// TwinCAT 3 PLC project drivePLC
// ProgramVersion: 3.1.4022.4
// libraries:
//   Tc2_MC2, * (Beckhoff Automation GmbH)
//   Tc2_NC, * (Beckhoff Automation GmbH)
//   Tc2_Standard, * (Beckhoff Automation GmbH)
//   Tc2_System, * (Beckhoff Automation GmbH)
//   Tc3_MC2_AdvancedHoming, * (Beckhoff Automation GmbH)
//   Tc3_Module, * (Beckhoff Automation GmbH)
//   VisuDialogs, * (System)
// project tree:
//   DUTs/ eLimitCoupling.TcDUT (not stored), eMcCommand.TcDUT (not stored), eRWParameter.TcDUT (not stored), ST_AxisControl.TcDUT, ST_MasterAxis.TcDUT (not stored), ST_MasterCoupling.TcDUT (not stored), ST_SimulateStage.TcDUT (not stored)
//   / GlobalTextList.TcGTLO, PlcTask.TcTTO, Visualization Manager.TcVMO (not stored)
//   GVLs/ GVL.TcGVL, Limits.TcGVL
//   POUs/ FB_AxisDrive.TcPOU, MAIN.TcPOU
//   VISUs/ Main.TcVIS
//   VISUs/Panels/ ButtonStates.TcTLO (not stored), CommandList.TcTLO (not stored), ImagePool.TcIPO (not stored), IO.TcVIS (not stored), SlitSet.TcVIS (not stored), Visualization.TcVIS
//   VISUs/Panels/Command VISUs/ AxisSimulation.TcVIS (not stored), Gearing.TcVIS (not stored), Homing.TcVIS (not stored), Parameters.TcVIS (not stored)
// real-time tasks:
//   TASK PlcTask: cycle T#10ms, priority 20, ADS port 350
// motion (NC):
//   TASK NC-Task 1 SAF: cycle T#2ms, priority 4, ADS port 501
//   TASK NC-Task 1 SVB: cycle T#10ms, priority 8, ADS port 511
//   AXIS North Blade (id 1)
//     Dynamic: AccelerationMaximum=5000, DecelerationMaximum=5000, Acceleration=10.7143, Deceleration=10.7143, Jerk=45.9184
//     Velo: RefSearch=1, RefSync=1, SlowManual=1, FastManual=3, Maximum=5
//     OtherSettings: AllowMotionCmdToSlave=true, DataPersistence=true, PulseDistancePos=0.1, PulseDistanceNeg=0.1
//     encoder EncType=19
//       EncPara: ScaleFactorNumerator=1, ScaleFactorDenominator=1048576, MaxCount=#xffffffff, ReferenceSystem=4
//         SoftEndMinControl: Range=-5
//         SoftEndMaxControl: Range=45
//         Inc: RefSearchInverse=true, RefSyncInverse=false, RefSoftSyncMask=#x0000ffff
//     drive DrvType=24
//       DrvPara: Inverse=true
//         Analog: VeloReferenz=5, ScaleFactorActTorque=0.1
//         TimeComp: TaskDelayCycles=1
//     controller CtrType=1
//       CtrPara: PriorControlFactor=1
//         PosDiffControl: Range=1
//         Observer: BandWidth=20
//   AXIS South Blade (id 2)
//     Dynamic: AccelerationMaximum=1500, DecelerationMaximum=1500, Acceleration=150, Deceleration=150, Jerk=225
//     Velo: RefSearch=1, RefSync=1, SlowManual=1, FastManual=3, Maximum=5
//     OtherSettings: AllowMotionCmdToSlave=true, DataPersistence=true, PulseDistancePos=0.1, PulseDistanceNeg=0.1
//     encoder EncType=19
//       EncPara: ScaleFactorNumerator=1, ScaleFactorDenominator=1048576, MaxCount=#xffffffff, ReferenceSystem=4
//         SoftEndMinControl: Range=-45
//         SoftEndMaxControl: Range=5
//         Inc: RefSoftSyncMask=#x0000ffff
//     drive DrvType=24
//       DrvPara: Inverse=true
//         Analog: VeloReferenz=5, ScaleFactorActTorque=0.1
//         TimeComp: TaskDelayCycles=1
//     controller CtrType=1
//       CtrPara: PriorControlFactor=1
//         PosDiffControl: Range=1
//         Observer: BandWidth=20
//   AXIS East Blade (id 3)
//     Dynamic: AccelerationMaximum=1500, DecelerationMaximum=1500, Acceleration=150, Deceleration=150, Jerk=225
//     Velo: RefSearch=1, RefSync=1, SlowManual=1, FastManual=3, Maximum=5
//     OtherSettings: AllowMotionCmdToSlave=true, DataPersistence=true, PulseDistancePos=0.1, PulseDistanceNeg=0.1
//     encoder EncType=19
//       EncPara: ScaleFactorNumerator=1, ScaleFactorDenominator=1048576, Inverse=true, MaxCount=#xffffffff, ReferenceSystem=4
//         SoftEndMinControl: Range=-5
//         SoftEndMaxControl: Range=45
//         Inc: RefSoftSyncMask=#x0000ffff
//     drive DrvType=24
//       Analog: VeloReferenz=5, ScaleFactorActTorque=0.1
//       TimeComp: TaskDelayCycles=1
//     controller CtrType=1
//       CtrPara: PriorControlFactor=1
//         PosDiffControl: Range=1
//         Observer: BandWidth=20
//   AXIS West Blade (id 4)
//     Dynamic: AccelerationMaximum=1500, DecelerationMaximum=1500, Acceleration=150, Deceleration=150, Jerk=225
//     Velo: RefSearch=1, RefSync=1, SlowManual=1, FastManual=3, Maximum=5
//     OtherSettings: AllowMotionCmdToSlave=true, DataPersistence=true, PulseDistancePos=0.1, PulseDistanceNeg=0.1
//     encoder EncType=19
//       EncPara: ScaleFactorNumerator=1, ScaleFactorDenominator=1048576, Inverse=true, MaxCount=#xffffffff, ReferenceSystem=4
//         SoftEndMinControl: Range=5
//         SoftEndMaxControl: Range=-45
//         Inc: RefSoftSyncMask=#x0000ffff
//     drive DrvType=24
//       Analog: VeloReferenz=5, ScaleFactorActTorque=0.1
//       TimeComp: TaskDelayCycles=1
//     controller CtrType=1
//       CtrPara: PriorControlFactor=1
//         Observer: BandWidth=20
//   AXIS VG (id 5)
//     Dynamic: AccelerationMaximum=200, DecelerationMaximum=200, Acceleration=150, Deceleration=150, Jerk=225
//     Velo: RefSearch=1, RefSync=1, SlowManual=1, FastManual=3, Maximum=3
//     OtherSettings: AllowMotionCmdToSlave=true, PulseDistancePos=0.1, PulseDistanceNeg=0.1
//     encoder EncType=1
//     drive DrvType=5
//       Analog: ScaleFactorActTorque=0.1
//       TimeComp: TaskDelayCycles=1
//     controller CtrType=1
//       CtrPara: PriorControlFactor=1
//         Observer: BandWidth=20
//   AXIS VC (id 6)
//     Dynamic: AccelerationMaximum=200, DecelerationMaximum=200, Acceleration=150, Deceleration=150, Jerk=225
//     Velo: RefSearch=1, RefSync=1, SlowManual=1, FastManual=3, Maximum=3
//     OtherSettings: AllowMotionCmdToSlave=true, PulseDistancePos=0.1, PulseDistanceNeg=0.1
//     encoder EncType=1
//     drive DrvType=5
//       Analog: ScaleFactorActTorque=0.1
//       TimeComp: TaskDelayCycles=1
//     controller CtrType=1
//       CtrPara: PriorControlFactor=1
//         Observer: BandWidth=20
//   AXIS HG (id 7)
//     Dynamic: AccelerationMaximum=200, DecelerationMaximum=200, Acceleration=150, Deceleration=150, Jerk=225
//     Velo: RefSearch=1, RefSync=1, SlowManual=1, FastManual=3, Maximum=3
//     OtherSettings: AllowMotionCmdToSlave=true, PulseDistancePos=0.1, PulseDistanceNeg=0.1
//     encoder EncType=1
//     drive DrvType=5
//       Analog: ScaleFactorActTorque=0.1
//       TimeComp: TaskDelayCycles=1
//     controller CtrType=1
//       CtrPara: PriorControlFactor=1
//         Observer: BandWidth=20
//   AXIS HC (id 8)
//     Dynamic: AccelerationMaximum=200, DecelerationMaximum=200, Acceleration=150, Deceleration=150, Jerk=225
//     Velo: RefSearch=1, RefSync=1, SlowManual=1, FastManual=3, Maximum=3
//     OtherSettings: AllowMotionCmdToSlave=true, PulseDistancePos=0.1, PulseDistanceNeg=0.1
//     encoder EncType=1
//     drive DrvType=5
//       Analog: ScaleFactorActTorque=0.1
//       TimeComp: TaskDelayCycles=1
//     controller CtrType=1
//       CtrPara: PriorControlFactor=1
//         Observer: BandWidth=20
// I/O:
//   DEVICE Device 1 (EtherCAT), AmsNetId 5.60.136.192.2.1
//     Term 1 (EK1200) [EK1200-5000 EtherCAT Power supply (2A E-Bus)]
//       Limits Output (EL2008) [EL2008 8Ch. Dig. Output 24V, 0.5A]
//       Limits Input (EL1008) [EL1008 8Ch. Dig. Input 24V, 3ms]
//       FB01 NORTH (EL7201) [EL7201 1Ch. MDP742 Servo motor output stage (50V, 4A)]
//       FB02 SOUTH (EL7201) [EL7201 1Ch. MDP742 Servo motor output stage (50V, 4A)]
//       FB03 EAST (EL7201) [EL7201 1Ch. MDP742 Servo motor output stage (50V, 4A)]
//       FB04 WEST (EL7201) [EL7201 1Ch. MDP742 Servo motor output stage (50V, 4A)]
//       DR01 NORTH (EL7047) [EL7047 1Ch. Stepper motor output stage (50V, 5A)]
//       DR02  SOUTH (EL7047) [EL7047 1Ch. Stepper motor output stage (50V, 5A)]
//       DR03 EAST (EL7047) [EL7047 1Ch. Stepper motor output stage (50V, 5A)]
//       DR04 WEST (EL7047) [EL7047 1Ch. Stepper motor output stage (50V, 5A)]
//       Term 21 (EL9011) [EL9011 End Terminal]
//   DEVICE Device 4 (COM Port)
// variable links:
//   NC-Task 1 SAF/Axes/East Blade <-> Device 1 (EtherCAT)/Term 1 (EK1200)/DR03 EAST (EL7047)
//     Drive/Inputs/In/nState1 @bit 3 <-> STM Status/Status/Error
//     Drive/Inputs/In/nState1 @bit 7 <-> STM Status/Status/Motor stall
//     Drive/Inputs/In/nState1 @bit 5 <-> STM Status/Status/Moving negative
//     Drive/Inputs/In/nState1 @bit 4 <-> STM Status/Status/Moving positive
//     Drive/Inputs/In/nState1 @bit 1 <-> STM Status/Status/Ready
//     Drive/Inputs/In/nState1 <-> STM Status/Status/Ready to enable
//     Drive/Inputs/In/nState1 @bit 6 <-> STM Status/Status/Torque reduced
//     Drive/Inputs/In/nState1 @bit 2 <-> STM Status/Status/Warning
//     Drive/Inputs/In/nState2 @bit 3 <-> STM Status/Status/Digital input 1
//     Drive/Inputs/In/nState2 @bit 4 <-> STM Status/Status/Digital input 2
//     Drive/Inputs/In/nState2 @bit 5 <-> STM Status/Status/Sync error
//     Drive/Inputs/In/nState2 @bit 7 <-> STM Status/Status/TxPDO Toggle
//     Drive/Inputs/In/nState4 @bit 1 <-> WcState/InputToggle
//     Drive/Inputs/In/nState4 <-> WcState/WcState
//     Drive/Outputs/Out/nCtrl1 <-> STM Control/Control/Enable
//     Drive/Outputs/Out/nCtrl1 @bit 2 <-> STM Control/Control/Reduce torque
//     Drive/Outputs/Out/nCtrl1 @bit 1 <-> STM Control/Control/Reset
//     Drive/Outputs/Out/nCtrl2 @bit 3 <-> STM Control/Control/Digital output 1
//     Drive/Outputs/Out/nDataOut2[0] <-> STM Velocity/Velocity
//   NC-Task 1 SAF/Axes/East Blade <-> Device 1 (EtherCAT)/Term 1 (EK1200)/FB03 EAST (EL7201)
//     East Bladenc/Inputs/In/nDataIn1 <-> FB Position/Position
//     East Bladenc/Inputs/In/nDcInputTime <-> InfoData/DcInputShift
//     East Bladenc/Inputs/In/nState4 @bit 1 <-> WcState/InputToggle
//     East Bladenc/Inputs/In/nState4 <-> WcState/WcState
//   NC-Task 1 SAF/Axes/North Blade <-> Device 1 (EtherCAT)/Term 1 (EK1200)/DR01 NORTH (EL7047)
//     Drive/Inputs/In/nState1 @bit 3 <-> STM Status/Status/Error
//     Drive/Inputs/In/nState1 @bit 7 <-> STM Status/Status/Motor stall
//     Drive/Inputs/In/nState1 @bit 5 <-> STM Status/Status/Moving negative
//     Drive/Inputs/In/nState1 @bit 4 <-> STM Status/Status/Moving positive
//     Drive/Inputs/In/nState1 @bit 1 <-> STM Status/Status/Ready
//     Drive/Inputs/In/nState1 <-> STM Status/Status/Ready to enable
//     Drive/Inputs/In/nState1 @bit 6 <-> STM Status/Status/Torque reduced
//     Drive/Inputs/In/nState1 @bit 2 <-> STM Status/Status/Warning
//     Drive/Inputs/In/nState2 @bit 3 <-> STM Status/Status/Digital input 1
//     Drive/Inputs/In/nState2 @bit 4 <-> STM Status/Status/Digital input 2
//     Drive/Inputs/In/nState2 @bit 5 <-> STM Status/Status/Sync error
//     Drive/Inputs/In/nState2 @bit 7 <-> STM Status/Status/TxPDO Toggle
//     Drive/Inputs/In/nState4 @bit 1 <-> WcState/InputToggle
//     Drive/Inputs/In/nState4 <-> WcState/WcState
//     Drive/Outputs/Out/nCtrl1 <-> STM Control/Control/Enable
//     Drive/Outputs/Out/nCtrl1 @bit 2 <-> STM Control/Control/Reduce torque
//     Drive/Outputs/Out/nCtrl1 @bit 1 <-> STM Control/Control/Reset
//     Drive/Outputs/Out/nCtrl2 @bit 3 <-> STM Control/Control/Digital output 1
//     Drive/Outputs/Out/nDataOut2[0] <-> STM Velocity/Velocity
//   NC-Task 1 SAF/Axes/North Blade <-> Device 1 (EtherCAT)/Term 1 (EK1200)/FB01 NORTH (EL7201)
//     Enc/Inputs/In/nDataIn1 <-> FB Position/Position
//     Enc/Inputs/In/nDcInputTime <-> InfoData/DcInputShift
//     Enc/Inputs/In/nState4 @bit 1 <-> WcState/InputToggle
//     Enc/Inputs/In/nState4 <-> WcState/WcState
//   NC-Task 1 SAF/Axes/South Blade <-> Device 1 (EtherCAT)/Term 1 (EK1200)/DR02  SOUTH (EL7047)
//     Drive/Inputs/In/nState1 @bit 3 <-> STM Status/Status/Error
//     Drive/Inputs/In/nState1 @bit 7 <-> STM Status/Status/Motor stall
//     Drive/Inputs/In/nState1 @bit 5 <-> STM Status/Status/Moving negative
//     Drive/Inputs/In/nState1 @bit 4 <-> STM Status/Status/Moving positive
//     Drive/Inputs/In/nState1 @bit 1 <-> STM Status/Status/Ready
//     Drive/Inputs/In/nState1 <-> STM Status/Status/Ready to enable
//     Drive/Inputs/In/nState1 @bit 6 <-> STM Status/Status/Torque reduced
//     Drive/Inputs/In/nState1 @bit 2 <-> STM Status/Status/Warning
//     Drive/Inputs/In/nState2 @bit 3 <-> STM Status/Status/Digital input 1
//     Drive/Inputs/In/nState2 @bit 4 <-> STM Status/Status/Digital input 2
//     Drive/Inputs/In/nState2 @bit 5 <-> STM Status/Status/Sync error
//     Drive/Inputs/In/nState2 @bit 7 <-> STM Status/Status/TxPDO Toggle
//     Drive/Inputs/In/nState4 @bit 1 <-> WcState/InputToggle
//     Drive/Inputs/In/nState4 <-> WcState/WcState
//     Drive/Outputs/Out/nCtrl1 <-> STM Control/Control/Enable
//     Drive/Outputs/Out/nCtrl1 @bit 2 <-> STM Control/Control/Reduce torque
//     Drive/Outputs/Out/nCtrl1 @bit 1 <-> STM Control/Control/Reset
//     Drive/Outputs/Out/nCtrl2 @bit 3 <-> STM Control/Control/Digital output 1
//     Drive/Outputs/Out/nDataOut2[0] <-> STM Velocity/Velocity
//   NC-Task 1 SAF/Axes/South Blade <-> Device 1 (EtherCAT)/Term 1 (EK1200)/FB02 SOUTH (EL7201)
//     Enc/Inputs/In/nDataIn1 <-> FB Position/Position
//     Enc/Inputs/In/nDcInputTime <-> InfoData/DcInputShift
//     Enc/Inputs/In/nState4 @bit 1 <-> WcState/InputToggle
//     Enc/Inputs/In/nState4 <-> WcState/WcState
//   NC-Task 1 SAF/Axes/West Blade <-> Device 1 (EtherCAT)/Term 1 (EK1200)/DR04 WEST (EL7047)
//     Drive/Inputs/In/nState1 @bit 3 <-> STM Status/Status/Error
//     Drive/Inputs/In/nState1 @bit 7 <-> STM Status/Status/Motor stall
//     Drive/Inputs/In/nState1 @bit 5 <-> STM Status/Status/Moving negative
//     Drive/Inputs/In/nState1 @bit 4 <-> STM Status/Status/Moving positive
//     Drive/Inputs/In/nState1 @bit 1 <-> STM Status/Status/Ready
//     Drive/Inputs/In/nState1 <-> STM Status/Status/Ready to enable
//     Drive/Inputs/In/nState1 @bit 6 <-> STM Status/Status/Torque reduced
//     Drive/Inputs/In/nState1 @bit 2 <-> STM Status/Status/Warning
//     Drive/Inputs/In/nState2 @bit 3 <-> STM Status/Status/Digital input 1
//     Drive/Inputs/In/nState2 @bit 4 <-> STM Status/Status/Digital input 2
//     Drive/Inputs/In/nState2 @bit 5 <-> STM Status/Status/Sync error
//     Drive/Inputs/In/nState2 @bit 7 <-> STM Status/Status/TxPDO Toggle
//     Drive/Inputs/In/nState4 @bit 1 <-> WcState/InputToggle
//     Drive/Inputs/In/nState4 <-> WcState/WcState
//     Drive/Outputs/Out/nCtrl1 <-> STM Control/Control/Enable
//     Drive/Outputs/Out/nCtrl1 @bit 2 <-> STM Control/Control/Reduce torque
//     Drive/Outputs/Out/nCtrl1 @bit 1 <-> STM Control/Control/Reset
//     Drive/Outputs/Out/nCtrl2 @bit 3 <-> STM Control/Control/Digital output 1
//     Drive/Outputs/Out/nDataOut2[0] <-> STM Velocity/Velocity
//   NC-Task 1 SAF/Axes/West Blade <-> Device 1 (EtherCAT)/Term 1 (EK1200)/FB04 WEST (EL7201)
//     Enc/Inputs/In/nDataIn1 <-> FB Position/Position
//     Enc/Inputs/In/nDcInputTime <-> InfoData/DcInputShift
//     Enc/Inputs/In/nState4 @bit 1 <-> WcState/InputToggle
//     Enc/Inputs/In/nState4 <-> WcState/WcState
//   drivePLC/drivePLC Instance <-> Device 1 (EtherCAT)/Term 1 (EK1200)/Limits Input (EL1008)
//     PlcTask Inputs/Limits.BwLimit[1] <-> Channel 2/NORTH CENTRE
//     PlcTask Inputs/Limits.BwLimit[2] <-> Channel 4/SOUTH OPEN
//     PlcTask Inputs/Limits.BwLimit[3] <-> Channel 5/EAST CENTRE
//     PlcTask Inputs/Limits.BwLimit[4] <-> Channel 7/WEST OPEN
//     PlcTask Inputs/Limits.FwLimit[1] <-> Channel 1/NORTH OPEN
//     PlcTask Inputs/Limits.FwLimit[2] <-> Channel 3/SOUTH CENTRE
//     PlcTask Inputs/Limits.FwLimit[3] <-> Channel 6/EAST OPEN
//     PlcTask Inputs/Limits.FwLimit[4] <-> Channel 8/WEST CENTRE
//   drivePLC/drivePLC Instance <-> Device 1 (EtherCAT)/Term 1 (EK1200)/Limits Output (EL2008)
//     PlcTask Outputs/MAIN.limitEnable1 <-> Channel 1/NORTH/SOUTH LIMITS
//     PlcTask Outputs/MAIN.limitEnable2 <-> Channel 2/EAST/WEST LIMITS
//   drivePLC/drivePLC Instance <-> NC-Task 1 SAF/Axes/East Blade
//     PlcTask Inputs/GVL.axes[3].Axis.NcToPlc <-> Outputs/ToPlc
//     PlcTask Outputs/GVL.axes[3].Axis.PlcToNc <-> Inputs/FromPlc
//   drivePLC/drivePLC Instance <-> NC-Task 1 SAF/Axes/HC
//     PlcTask Inputs/GVL.axes[8].Axis.NcToPlc <-> Outputs/ToPlc
//     PlcTask Outputs/GVL.axes[8].Axis.PlcToNc <-> Inputs/FromPlc
//   drivePLC/drivePLC Instance <-> NC-Task 1 SAF/Axes/HG
//     PlcTask Inputs/GVL.axes[7].Axis.NcToPlc <-> Outputs/ToPlc
//     PlcTask Outputs/GVL.axes[7].Axis.PlcToNc <-> Inputs/FromPlc
//   drivePLC/drivePLC Instance <-> NC-Task 1 SAF/Axes/North Blade
//     PlcTask Inputs/GVL.axes[1].Axis.NcToPlc <-> Outputs/ToPlc
//     PlcTask Outputs/GVL.axes[1].Axis.PlcToNc <-> Inputs/FromPlc
//   drivePLC/drivePLC Instance <-> NC-Task 1 SAF/Axes/South Blade
//     PlcTask Inputs/GVL.axes[2].Axis.NcToPlc <-> Outputs/ToPlc
//     PlcTask Outputs/GVL.axes[2].Axis.PlcToNc <-> Inputs/FromPlc
//   drivePLC/drivePLC Instance <-> NC-Task 1 SAF/Axes/VC
//     PlcTask Inputs/GVL.axes[6].Axis.NcToPlc <-> Outputs/ToPlc
//     PlcTask Outputs/GVL.axes[6].Axis.PlcToNc <-> Inputs/FromPlc
//   drivePLC/drivePLC Instance <-> NC-Task 1 SAF/Axes/VG
//     PlcTask Inputs/GVL.axes[5].Axis.NcToPlc <-> Outputs/ToPlc
//     PlcTask Outputs/GVL.axes[5].Axis.PlcToNc <-> Inputs/FromPlc
//   drivePLC/drivePLC Instance <-> NC-Task 1 SAF/Axes/West Blade
//     PlcTask Inputs/GVL.axes[4].Axis.NcToPlc <-> Outputs/ToPlc
//     PlcTask Outputs/GVL.axes[4].Axis.PlcToNc <-> Inputs/FromPlc

CONFIGURATION drivePLC
    RESOURCE PLC ON TwinCAT3
        TASK PlcTask(INTERVAL := T#10ms, PRIORITY := 20);
        PROGRAM MAIN WITH PlcTask : MAIN;
    END_RESOURCE
END_CONFIGURATION

// ---- DUTs/ST_AxisControl.TcDUT
{attribute 'OPC.UA.DA' := '1'}
TYPE ST_AxisControl :
STRUCT
	//OPC UA functionality not implemented yet
	(*For a list of parameters required to operate each motion control funciton block
	see the DUT eMcCommand*)
	
	bExecute			:	BOOL;			//Rising edge to execute command
	bReset				:	BOOL;			//Reset axis signal, must be combined with other signals
	eCommand			:	eMcCommand;		//Motion command for axis
	bEnable				: 	BOOL;			//Controller enable
	fOverride			:	LREAL;			//Controller override %
	fVelocity			:	LREAL;			//Velocity must be specified, no default used
	fAcceleration		:	LREAL;			//Not all FBs use, need to change this, 0 is NC default
	fDeceleration		:	LREAL;			//Not all FBs use, need to change this, 0 is NC default
	fDistance			:	LREAL;			//Used for relative positioning
	fPosition			:	LREAL;			//Used for absolute positioning	
	bJogForward			:	BOOL;			//Jog forward
	bJogBackward		:	BOOL;			//Jog backward
	
	bInput				:	BOOL;			//Generic input that is utilised to control some functionality
	
	bSoftLimPosEn		:	BOOL;			//Enable/disable positive direction software limit
	bSoftLimNegEn		:	BOOL;			//Enable/disable negative direction software limit
	bPosLagEn			:	BOOL;			//Enable/disable position lag
	
	fActPosition		:	LREAL;
	fActVelocity		:	LREAL;
	bNegativeDirection	:	BOOL;
	bPositiveDirection	:	BOOL;
	bCalibrated			:	BOOL;
	
	//Gearing parameters
	masterAxis			:	UINT:=1;						//Axes[ ] index for master		- GearIn
	fGearRatioNum		:	LREAL;							//GearIn ratio numerator
	iGearRatioDen		:	UINT;							//GearIn ratio denominator
	masterAxes			:	ARRAY[1..4] OF ST_MasterAxis;	//ST to hold index and ratio for masters 	- GearInMultiMaster
	
	//NC Parameters	
	iParameterIndex		:	INT;					//Index for checking parameters
	fParameterValue		:	LREAL;					//Holder for assigning new values
	fParameters			:	ARRAY [1..17] OF LREAL;	//Array to hold NC parameters
	
	//MISC
	sAxisName			:	STRING;					//User set name string for axis
	sAxisDesc			:	STRING;					//User set description string for axis
	
	//Outputs
	bFwEnabled			:	BOOL;					//Positive movement of axis is enabled/disabled
	bBwEnabled			:	BOOL;					//Negative movement of axis is enabled/disabled
	bAxisReady			:	BOOL;					//Output of McPower block	
	bError				:	BOOL;					//Motion function block has produced error (NC drive not necessarily in error state)
	iErrorID			:	UDINT;					//Motion function block errorID				
	bBusy				:	BOOL;					//Axis busy
	bMoving				:	BOOL;					//Axis moving					
	bDone				:	BOOL;					//Last function block executed successfully			
	
	iAxisState			:	UINT;					//PLC Open NC statemachine, int assigned to individual NC bool state outputs
	(*	100 - Disabled
		200 - Standstill
		300 - Homing
		400 - Discrete Motion
		500 - Synchronized Motion
		600 - Continuous Motion
		700 - Stopping
		999 - Error
	*)
	
	buffer				:	MC_BufferMode	:=	MC_Aborting;							//Placeholder - Not currently used
	
	//Homing
	fHomeVelocity		:	LREAL	:=1;							//Homing routine velocity 							- initialised for testing purposes
	fHomeTorque			:	LREAL;									//Homing torque limit (not all drives support this)
	fHomePosition		:	LREAL;									//Position set at NC when homing step finished
	fHomeDistance		:	LREAL;									//Relative distance to move after homing
	tHomeTimeLimit		:	TIME:=T#60S;							//Homing timeout limit, FB errors is exceeded 		- initialised for testing purposes
	fHomeDistanceLimit	:	LREAL:=2000;							//Homing distance limit, FB errors if exceeded 		- initialised for testing purposes
	
	MCHomeDirection		:	MC_Home_Direction:=	mcSwitchPositive;	(*~ (OPC:0:not available) *)
	(*	Direction to begin homing. Not all are compatible with every advanced homing step
		mcPositiveDirection	-	always start positive
		mcNegativeDirection	-	always start negative
		mcSwitchPositive	-	start positive unless already on the switch
		mcSwitchNegative	-	start negative unless already on the switch
		
	*)
	

	MCSwitchMode		:	MC_Switch_Mode:= mcRisingEdge;			(*~ (OPC:0:not available) *)
	(* Switch detection behaviour, I am not entirely convinced these are all working as they are meant to, further work required. Not all detection methods work with every 
	step either so they have to be updated.
		mcOn
		mcOff
		mcRisingEdge
		mcFallingEdge
		mcEdgeSwitchPositive
		mcEdgeSwitchNegative
		mcRisingEdgeInverse
		mcFallingEdgeInverse	
	*)

	MCSignalRef			:	MC_Ref_Signal_Ref;		(*~ (OPC:0:not available) *)
	
	(*Further investigation required on how exactly this MCSignalRef works, it seems to contain signalsource, touch probe and level signals,
	my current understanding is that with physical hardware connected the MCSignalRef signal source should default to the NC hardware so nothing has to be linked
	for the encoder index, however the source may need to be changed for the absSwitch homing which would just require an additional line of code in the driveFB step command
	I also do not have any bool available for linking an absolute switch to an axis at the moment

		SignalSource : E_SignalSource := SignalSource_Default;
		TouchProbe : E_TouchProbe := PlcEvent;
		Level : BOOL;
	*)

	Axis				:	AXIS_REF;	(*~ (OPC:0:not available) *)

END_STRUCT
END_TYPE

// ---- GVLs/GVL.TcGVL
{attribute 'qualified_only'}
VAR_GLOBAL
	iAxis		:	UINT;												//Indexing variable for exposing which axis currently being run though drive function block
	axes			:	ARRAY [1..GVL.axisNumMax] OF ST_AxisControl; 	(*~ (OPC: 1 : available for OPC-clients)*)
	
//HMI Parameters	-	These can hopefully be removed on upgrading to the new HMI tool
	SwLimitPos	:	LREAL;
	SwLimitNeg	:	LREAL;
	MaxPositionLag	:	LREAL;
	MaxVelocityAppl	:	LREAL;
	MaxAccelerationAppl	:	LREAL;
	MaxDecelerationAppl	:	LREAL;
	MaxJerkAppl			:	LREAL;
	
END_VAR
VAR_GLOBAL CONSTANT
	axisNumMax	:	UINT:=8;
	axisCoupleMax	:	UINT:=4;
END_VAR

// ---- GVLs/Limits.TcGVL
{attribute 'qualified_only'}
VAR_GLOBAL
	FwLimit				AT	%I*	: ARRAY[1..GVL.axisNumMax] OF BOOL;		(*~ (OPC: 1 : available for OPC-clients) (OPC_PROP[0005]: 1 : OPC_PROP_RIGHTS, here read/write) *)
	BwLimit				AT  %I*	: ARRAY[1..GVL.axisNumMax] OF BOOL;		(*~ (OPC: 1 : available for OPC-clients) (OPC_PROP[0005]: 1 : OPC_PROP_RIGHTS, here read/write) *)
	
	coupledFwLimit		: ARRAY [1..GVL.axisNumMax] OF ARRAY [1..5] OF ST_MasterCoupling;	//Store for slave/master linking
	coupledBwLimit		: ARRAY [1..GVL.axisNumMax] OF ARRAY [1..5] OF ST_MasterCoupling;	//Store for slave/master linking

END_VAR

// ---- POUs/MAIN.TcPOU
PROGRAM MAIN
VAR
	{attribute 'OPC.UA.DA' := '1'}
	{attribute 'OPC.UA.DA.StructuredType' := '1'}
	//Simulate virtual axes
	simulated		:	ARRAY [1..GVL.axisNumMax] OF ST_SimulateStage;
	bSimulate		:	ARRAY [1..GVL.axisNumMax] OF BOOL;	//Do we want to simulate?
	
	//{attribute 'OPC.UA.DA' := '0'}
	drives			:	ARRAY [1..GVL.axisNumMax] OF FB_AxisDrive;	
	
	bDisableMC		:	BOOL; 		//boolean control if true the motion control application specific code is disabled - dumb box
	iState			:	UINT;		//state machine index

	(*
		Outputs that are set in the hmi and wired to power axis limit switches. Currently not configred as part of the programme
		Will be added to ST_AxisControl in future
	*)
	limitEnable1	AT %Q*	: BOOL;
	limitEnable2	AT %Q*	: BOOL;	
	
	i: UINT;		//General indexing value for FOR loops	
	
	//HMI VARIABLES	
	hmiAxisSelect	:	UINT:=1;

END_VAR

AXES();
PROG();
//SIMULATE();

ACTION AXES:
FOR GVL.iAxis:=1 TO GVL.axisNumMax DO
	drives[GVL.iAxis](AxisController:=GVL.axes[GVL.iAxis]);
END_FOR
END_ACTION

(*
	Scans through axes (from low to high) checking "done" status
*)
METHOD CheckCoupled : BOOL
VAR_INPUT
	iLow	:	UINT;		//lowest index to check
	iHigh	:	UINT;		//highest index to check
END_VAR

VAR
	i		:	UINT;
END_VAR
CheckCoupled:=TRUE;
FOR i:=iLow TO iHigh BY 1 DO
	CheckCoupled:= CheckCoupled AND (GVL.axes[i].iAxisState=500);
END_FOR
END_METHOD

(*
	Scans through axes (from low to high) checking "done" status
*)
METHOD CheckDone : BOOL
VAR_INPUT
	iLow	:	UINT;		//lowest index to check
	iHigh	:	UINT;		//highest index to check
END_VAR

VAR
	i		:	UINT;
END_VAR
CheckDone:=TRUE;
FOR i:=iLow TO iHigh BY 1 DO
	CheckDone:= CheckDone AND GVL.axes[i].bDone;
END_FOR
END_METHOD

(*
	Scans through axes (from low to high) checking "done" status
*)
METHOD CheckMoving : BOOL
VAR_INPUT
	iLow	:	UINT;		//lowest index to check
	iHigh	:	UINT;		//highest index to check
END_VAR

VAR
	i		:	UINT;
	statiks: INT;
END_VAR
CheckMoving:=FALSE;
FOR i:=iLow TO iHigh BY 1 DO
	CheckMoving:= CheckMoving OR (GVL.axes[i].Axis.status.Moving);
END_FOR
END_METHOD

(*
	Gear out an axis
*)
METHOD GearOut : BOOL
VAR_INPUT
	i	:	UINT;	//Axis index to gear out
END_VAR
GVL.axes[i].eCommand:=eMcCommand.GearOut;
GVL.axes[i].bExecute:=TRUE;
END_METHOD

(*
	Power up a single axis of index i
*)
METHOD PowerUp : BOOL
VAR_INPUT
	i	:	UINT;
END_VAR
GVL.axes[i].bEnable:=TRUE;
GVL.axes[i].fOverride:=100;
Limits.FwLimit[i]:=TRUE;	//Set high as I have no hardware linked
Limits.BwLimit[i]:=TRUE;	//Set high as I have no hardware linked
END_METHOD

ACTION PROG:
CASE iState OF
	0:	//CHECK AXIS ID's are correct. Gearing limits currently requires the assigned array index of an axis to match the NC ID.
		//May be possible to negate this by changing axes to GVLs so that they can be seen within the drives function - CASE 0 NO LONGER REQ
		iState:=1;
		FOR i:=1 TO GVL.axisNumMax BY 1 DO
			IF GVL.axes[i].Axis.NcToPlc.AxisId <> i THEN
				iState:=999;
			END_IF
		END_FOR
		
	1:	//Gear out all axes to begin
		FOR i:=1 TO 8 BY 1 DO
			GearOut(i:=i);
		END_FOR
		iState:= 2;
	2:	//Wait for gear out
		IF CheckDone(iLow:=1, iHigh:=8) THEN
			iState:=3;
		END_IF
	3:	//Power up axes (and set limits true as no hardware connected)
		limitEnable1 	:=	TRUE;
		limitEnable2	:=	TRUE;
		FOR i:=1 TO 8 BY 1 DO
			PowerUp(i:=i);
		END_FOR
		iState:= 4;
		
	4:	//HOMING ROUTING
		
		iState:=	10;
		
		
	10:	//Start of main state loop. Are the blades coupled in to the virtual axes?
		//SlitPositions(North:=1,South:=2,East:=3,West:=4,VG:=5,VC:=6,HG:=7,HC:=8);
		IF NOT CheckCoupled(iLow:=1, iHigh:=4) THEN
			iState:=11;
		END_IF
		
	11:	//Blades are not coupled. Update the virtual positions
		FOR i:=1 TO 8 BY 1 DO
			GearOut(i:=i);
		END_FOR
	
		iState:=12;
			
		
	12:	//Confirm positions set
		IF CheckDone(iLow:=5,iHigh:=8) THEN
			iState:=12;
		END_IF	
		iState:=13;
	
	13:	//Check Moving
		SlitPositions(North:=1,South:=2,East:=3,West:=4,VG:=5,VC:=6,HG:=7,HC:=8);
		iState:=14;
		

	14: //Blades not moving, time to setup again
		IF CheckDone(iLow:=5,iHigh:=8) THEN
			iState:=15;
		END_IF			

		
	15:	//Check movin
		IF CheckMoving(iLow:=1, iHigh:=4) THEN
			iState:= 13;
		ELSE
			iState:=16;
		END_IF
	

	16:	//Multimaster gearin
		SlitSetup(North:=1,South:=2,East:=3,West:=4,VG:=5,VC:=6,HG:=7,HC:=8);
		iState:=17;	
		
	17:
		IF CheckDone(iLow:=1,iHigh:=8) THEN
			iState:=10;
		END_IF
		
	50:
		
	51:
						
			
	100:	//DO NOTHING

		
	
	999: //ERROR
		//INOP STATE	
END_CASE
END_ACTION

ACTION SIMULATE:
(*
Simulate axes if bool set TRUE
*)
FOR i:=1 TO GVL.axisNumMax BY 1 DO
	IF bSimulate[i] THEN
		simulateStage(position:=GVL.axes[i].Axis.NcToPlc.ActPos, iAxis:=i, simulated:=simulated[i]);
		GVL.axes[i].MCSignalRef.Level:=simulated[i].absSw;
	END_IF
END_FOR
END_ACTION

(*
	Basic virtual axis simulation.
	Will trigger limit switches beyond set points
	Will trigger absolute switch between given set points
*)
METHOD simulateStage : BOOL
VAR_INPUT
	position	:	LREAL;		//Axis current position
	iAxis		:	UINT;		//Axis index
END_VAR
VAR_IN_OUT
	simulated	:	ST_SimulateStage;	//Struct to hold simulation parameters
END_VAR
Limits.FwLimit[iAxis]:= position < simulated.fHighLim;
Limits.BwLimit[iAxis]:= position > simulated.fLowLim;

simulated.absSw:= (position < simulated.fHighAbs) AND (position > simulated.fLowAbs);
END_METHOD

(*
	Calculate gap positions of a slit set given N/S/E/W blades
*)
METHOD SlitPositions : BOOL
VAR_INPUT
	North	:	UINT;	//North blade index
	South	:	UINT;	//South blade index
	East	:	UINT;	//East blade index
	West	:	UINT;	//West blade index
	VG		:	UINT;	//Vertical gap size index
	VC		:	UINT;	//Vertical gap centre index
	HG		:	UINT;	//Horizontal gap size index
	HC		:	UINT;	//Horizontal gap centre index
END_VAR
GVL.axes[VG].eCommand:=eMcCommand.SetPosition;
GVL.axes[VG].fPosition:=GVL.axes[North].Axis.NcToPlc.ActPos-GVL.axes[South].Axis.NcToPlc.ActPos;
GVL.axes[VG].bExecute:=TRUE;

GVL.axes[VC].eCommand:=eMcCommand.SetPosition;
GVL.axes[VC].fPosition:=(GVL.axes[North].Axis.NcToPlc.ActPos+GVL.axes[South].Axis.NcToPlc.ActPos)/2;
GVL.axes[VC].bExecute:=TRUE;

GVL.axes[HG].eCommand:=eMcCommand.SetPosition;
GVL.axes[HG].fPosition:=GVL.axes[East].Axis.NcToPlc.ActPos-GVL.axes[West].Axis.NcToPlc.ActPos;
GVL.axes[HG].bExecute:=TRUE;

GVL.axes[HC].eCommand:=eMcCommand.SetPosition;
GVL.axes[HC].fPosition:=(GVL.axes[East].Axis.NcToPlc.ActPos+GVL.axes[West].Axis.NcToPlc.ActPos)/2;
GVL.axes[HC].bExecute:=TRUE;
END_METHOD

(*
	Gear in blades to gaps for a slit set
*)
METHOD SlitSetup : BOOL
VAR_INPUT
	North	:	UINT;
	South	:	UINT;
	East	:	UINT;
	West	:	UINT;
	VG		:	UINT;
	VC		:	UINT;
	HG		:	UINT;
	HC		:	UINT;
END_VAR
GVL.axes[North].eCommand:= eMcCommand.GearInMultiMaster;
GVL.axes[North].bExecute:=TRUE;
GVL.axes[NORTH].masterAxes[1].i:=VG;
GVL.axes[NORTH].masterAxes[2].i:=VC;
GVL.axes[NORTH].masterAxes[1].ratio:=0.5;
GVL.axes[NORTH].masterAxes[2].ratio:=1;

GVL.axes[South].eCommand:= eMcCommand.GearInMultiMaster;
GVL.axes[South].bExecute:=TRUE;
GVL.axes[South].masterAxes[1].i:=VG;
GVL.axes[South].masterAxes[2].i:=VC;
GVL.axes[South].masterAxes[1].ratio:=-0.5;
GVL.axes[South].masterAxes[2].ratio:=1;

GVL.axes[West].eCommand:= eMcCommand.GearInMultiMaster;
GVL.axes[West].bExecute:=TRUE;
GVL.axes[West].masterAxes[1].i:=HG;
GVL.axes[West].masterAxes[2].i:=HC;
GVL.axes[West].masterAxes[1].ratio:=-0.5;
GVL.axes[West].masterAxes[2].ratio:=1;


GVL.axes[East].eCommand:= eMcCommand.GearInMultiMaster;
GVL.axes[East].bExecute:=TRUE;
GVL.axes[East].masterAxes[1].i:=HG;
GVL.axes[East].masterAxes[2].i:=HC;
GVL.axes[East].masterAxes[1].ratio:=0.5;
GVL.axes[East].masterAxes[2].ratio:=1;
END_METHOD

END_PROGRAM

// ---- POUs/FB_AxisDrive.TcPOU
(*
	Function for motion control of single axis.
	Provides an interface to PLC Open motion control blocks.
	Controls linking of limit switches from slave to master axes.
*)
FUNCTION_BLOCK FB_AxisDrive
VAR_INPUT
END_VAR
VAR_IN_OUT
	AxisController		:	ST_AxisControl;
END_VAR
VAR_OUTPUT
END_VAR
VAR
	eCommandLatched		:	eMcCommand;		//Internally latched command signal, new commands cannot be issued until existing commands have completed.
	doneLatch	:	SR;						//Used to set done signal in AxisController DUT
	bDone		:	BOOL;					//Interal done flag which will be used for latching on an external done located in AxisController DUT
	iParam		:	INT:=1;					//index of NC parameters FBs, no 0 index on array so initialised to 1
	iIndex		:	UINT;					//index value used for limit coupling
	iMasterIndex		:	UINT;			//index value used for limit coupling
	
	//Boolean to store EnableFw and EnableBw of MCPower FB
	FwLimitsEnabled	:	BOOL;	
	BWLimitsEnabled	:	BOOL;
	
	mcDirection	:	MC_Direction;			//Direction control required in function blocks

(*
Motion Function blocks taken from the PLC OPEN standard as defined by PLC Open Standard
Function blocks commented out are yet to be added but the intention is to add these.
Those listed as //NOT IMPLEMENTED have come from the standard but Beckhoff do not support, 
these have been added just as a placeholder for future support.
*)
	//Not Implemented
	//MCReadDigitalInput		:	MC_ReadDigitalInput;			//NOT IMPLEMENTED		
	//MCReadDigitalOutput		:	MC_ReadDigitalOutput;			//NOT IMPLEMENTED	
	//MCWriteDigitalOutput		:	MC_WriteDigitalOutput;			//NOT IMPLEMENTED
	//MCReadActualTorque		:	MC_ReadActualTorque;			//NOT IMPLEMENTED	
	//MCReadAxisInfo			:	MC_ReadAxisInfo;				//NOT IMPLEMENTED	
	//MCReadMotionState			:	MC_ReadMotionState;				//NOT IMPLEMENTED
	//MCDigitalCamSwitch		:	MC_DigitalCamSwitch;			//NOT IMPLEMENTED
	//MCTorqueControl			:	MC_TorqueControl;				//NOT IMPLEMENTED		
	//MCPositionProfile			:	MC_PositionProfile;				//NOT IMPLEMENTED		
	//MCVelocityProfile			:	MC_VelocityProfile;				//NOT IMPLEMENTED		
	//MCAccelerationProfile		:	MC_AccelerationProfile;			//NOT IMPLEMENTED
	
	
	(* Administrative Function Blocks *)                                                                     
	MCReset						:	MC_Reset;											
	MCPower						:	MC_Power;										
	//MCReadStatus				:	MC_ReadStatus;					//Same as Axis.ReadStatus();						
	//MCReadAxisError			:	MC_ReadAxisError;									
	MCReadParameter				:	MC_ReadParameter;														
	MCWriteParameter			:	MC_WriteParameter;										
	MCWriteBoolParameter		:	MC_WriteBoolParameter;								
		
	//MCReadActualPosition		:	MC_ReadActualPosition;								
	//MCReadActualVelocity		:	MC_ReadActualVelocity;								
		
	MCSetPosition				:	MC_SetPosition;										
	//MCSetOverride				:	MC_SetOverride;										
	//MCTouchProbe				:	MC_TouchProbe;										
		
	//MCAbortTrigger			:	MC_AbortTrigger;									
	//MCAbortSuperposition		:	MC_AbortSuperposition;			//Listed as HaltSuperimposed in PLC Open standard	
	//MCCamTableSelect			:	MC_CamTableSelect;									
	
	(* Motion Function Blocks *)
	//MCHome					:	MC_Home;											
	MCJog						:	MC_Jog;												
	MCStop						:	MC_Stop;											
	//MCHalt					:	MC_Halt;											
	MCMoveAbsolute				:	MC_MoveAbsolute;									
	MCMoveRelative				:	MC_MoveRelative;									
	//MCMoveAdditive			:	MC_MoveAdditive;									
	//MCMoveSuperimposed		:	MC_MoveSuperimposed;								
	MCMoveVelocity				:	MC_MoveVelocity;									
	//MCMoveContinuousAbsolute	:	MC_MoveContinuousAbsolute;						
	//MCMoveContinuousRelative	:	MC_MoveContinuousRelative;						
	//MCMoveModulo				:	MC_MoveModulo;										
	
	(* Synchronised Motion Function Blocks *)		
	MCGearIn					:	MC_GearIn;											
	//MCGearInDyn				:	MC_GearInDyn;										
	MCGearInMultiMaster			:	MC_GearInMultiMaster;								
	MCGearOut					:	MC_GearOut;												                                                                                    
	//MCHaltPhasing				:	MC_HaltPhasing;										
	//MCPhasingAbsolute			:	MC_PhasingAbsolute;									
	//MCPhasingRelative			:	MC_PhasingRelative;										                                                                                                                                                 
	//MCCamIn					:	MC_CamIn;											
	//MCCamOut					:	MC_CamOut;											
	//MCCamScaling				:	MC_CamScaling;										                                                      
	//MCCamAdd					:	MC_CamAdd;											
	//MCCamExchange				:	MC_CamExchange;										
	//MCCamInV2					:	MC_CamIn_V2;		//REQUIRED FOR MULTICAMMING 	
	//MCCamRemove				:	MC_CamRemove;										
	//MCCamScalingV2			:	MC_CamScaling_V2;									

	(* Advanced Homing Steps and Finishing Moves *)
	MCFinishHoming			:	MC_FinishHoming;
	//MCHomeDirect			:	MC_HomeDirect;
	//MCAbortHoming			:	MC_AbortHoming;
	MCStepAbsoluteSwitch	:	MC_StepAbsoluteSwitch;
	//MCStepBlock			:	MC_StepBlock;
	//MCStepBlockLagBased	:	MC_StepBlockLagBased;
	//MCStepLimitSwitch		:	MC_StepLimitSwitch;
	//MCStepReferencePulse	:	MC_StepReferencePulse;
	
	
	(* Additional variable structures required for Advanced Homing *)
	//MCSignalRef			:	MC_Ref_Signal_Ref;
	StOptions				:	ST_Home_Options;
	StOptions2				:	ST_Home_Options2;
	StOptions3				:	ST_Home_Options3;
	StOptions4				:	ST_Home_Options4;
	MCHomingParameter		:	MC_HomingParameter;		//Must be passed between homing steps.		
							
		
END_VAR

AxisController.Axis.ReadStatus();
AxisController.fActPosition:= AxisController.Axis.NcToPlc.ActPos;
AxisController.fActVelocity:= AxisController.Axis.NcToPlc.ActVelo;
AxisController.bNegativeDirection:= AxisController.Axis.status.NegativeDirection;
AxisController.bPositiveDirection:= AxisController.Axis.Status.PositiveDirection;
AxisController.bCalibrated:= AxisController.Axis.Status.Homed;

//////////////////////////////////////////////////////////////////////
//     _   __  _____ ____    ____ _____  _  _____ _____ ____  		//
//    / \  \ \/ |_ _/ ___|  / ___|_   _|/ \|_   _| ____/ ___| 		//
//   / _ \  \  / | |\___ \  \___ \ | | / _ \ | | |  _| \___ \ 		//
//  / ___ \ /  \ | | ___) |  ___) || |/ ___ \| | | |___ ___) |		//
// /_/   \_/_/\_|___|____/  |____/ |_/_/   \_|_| |_____|____/ 		//
// 																	//
//////////////////////////////////////////////////////////////////////
                                                            
//Numerical representation for axis states - may use later for buffering functions.
IF AxisController.AXIS.Status.Disabled THEN
	AxisController.iAxisState:=		100;
ELSIF AxisController.AXIS.Status.StandStill THEN
	AxisController.iAxisState:=		200;
ELSIF AxisController.AXIS.Status.Homing	THEN
	AxisController.iAxisState:= 	300;
ELSIF AxisController.AXIS.Status.DiscreteMotion	THEN
	AxisController.iAxisState:=		400;
ELSIF AxisController.AXIS.Status.SynchronizedMotion	THEN
	AxisController.iAxisState:=		500;
ELSIF AxisController.AXIS.Status.ContinuousMotion	THEN
	AxisController.iAxisState:=		600;
ELSIF AxisController.AXIS.Status.Stopping	THEN
	AxisController.iAxisState:= 	700;	
ELSIF AxisController.AXIS.Status.Error THEN
	AxisController.iAxisState:=		999;	
ELSE
	AxisController.iAxisState:=		0;
END_IF

//////////////////////////////////////////////////////////////////////////////////////////
//  _     ___ __  __ ___ _____   ______        _____ _____ ____ _   _ _____ ____  		//
// | |   |_ _|  \/  |_ _|_   _| / ___\ \      / |_ _|_   _/ ___| | | | ____/ ___| 		//
// | |    | || |\/| || |  | |   \___ \\ \ /\ / / | |  | || |   | |_| |  _| \___ \ 		//
// | |___ | || |  | || |  | |    ___) |\ V  V /  | |  | || |___|  _  | |___ ___) |		//
// |_____|___|_|  |_|___| |_|   |____/  \_/\_/  |___| |_| \____|_| |_|_____|____/		//
//																						//
//////////////////////////////////////////////////////////////////////////////////////////

//Initialise Foward and Backward limits to the hardware limit switches for this axis
FwLimitsEnabled :=Limits.FwLimit[GVL.iAxis];
BwLimitsEnabled :=Limits.BwLimit[GVL.iAxis];

(*
Cycle through Limits.coupledFwLimit and Limits.coupledBwLimit.
Looking to see if any axes have the current axis (GVL.iAxis) listed as a master.
If this axis is listed as a master, check the hardware limits of that slave.
Gear ratio determines whether we are looking for a Forward or a Backward limit on the slave axis. 
If the limit switch is disabled, disable motion for this axis.
*)
FOR iIndex:=1 TO GVL.axisNumMax DO
	FOR iMasterIndex:=1 TO 5 DO
		//If listed as a master
		IF Limits.coupledFwLimit[iIndex][iMasterIndex].iMasterAxis = GVL.iAxis THEN
			//If forward limit linked to forward of slave, check forward limit of slave
			IF Limits.coupledFwLimit[iIndex][iMasterIndex].eLimitType=eLimitCoupling.FwSw AND NOT Limits.FwLimit[iIndex] THEN
				FwLimitsEnabled:=FALSE;
			END_IF
			//If forward limit linked to backwardof slave, check forward limit of slave
			IF Limits.coupledFwLimit[iIndex][iMasterIndex].eLimitType=eLimitCoupling.BwSw AND NOT Limits.BwLimit[iIndex] THEN
				FwLimitsEnabled:=FALSE;
			END_IF
			//If backward limit linked to forward of slave, check forward limit of slave
			IF Limits.coupledBwLimit[iIndex][iMasterIndex].eLimitType=eLimitCoupling.FwSw AND NOT Limits.FwLimit[iIndex] THEN
				BwLimitsEnabled:=FALSE;
			END_IF
			//If backward limit linked to backward of slave, check backward limit of slave
			IF Limits.coupledBwLimit[iIndex][iMasterIndex].eLimitType=eLimitCoupling.BwSw AND NOT Limits.BwLimit[iIndex] THEN
				BwLimitsEnabled:=FALSE;
			END_IF
		END_IF
	END_FOR
END_FOR

AxisController.bFwEnabled:=FwLimitsEnabled;		//Feedback to ST_AxisControl that forward positioning is available
AxisController.bBwEnabled:=BwLimitsEnabled;		//Feedback to ST_AxisControl that backward positioning is available

//////////////////////////////////////////////////////////
//  ____   _____        _______ ____    _   _ ____  	//
// |  _ \ / _ \ \      / | ____|  _ \  | | | |  _ \ 	//
// | |_) | | | \ \ /\ / /|  _| | |_) | | | | | |_) |	//
// |  __/| |_| |\ V  V / | |___|  _ <  | |_| |  __/ 	//
// |_|    \___/  \_/\_/  |_____|_| \_\  \___/|_|   		//
//														//
//////////////////////////////////////////////////////////
(*
Power up the axis.
Externally fed variables are bEnabled and fOverride, limits all controlled internally.
*)                                           
MCPower(
	Axis:=AxisController.Axis,
	Enable:=AxisController.bEnable,
	Enable_Positive:=FwLimitsEnabled,
	Enable_Negative:=BwLimitsEnabled,
	Override:=AxisController.fOverride,
	Status=>,
	Busy=>, 
	Active=>AxisController.bAxisReady,	//Maybe want a bPowered or bEnabled flag instead?
	Error=>,
	ErrorID=>
);

//////////////////////////////////////////////////////////////////////////////////////////////////////////
//  ____  _____    _    ____    ____   _    ____     _    __  __ _____ _____ _____ ____  ____  			//
// |  _ \| ____|  / \  |  _ \  |  _ \ / \  |  _ \   / \  |  \/  | ____|_   _| ____|  _ \/ ___| 			//
// | |_) |  _|   / _ \ | | | | | |_) / _ \ | |_) | / _ \ | |\/| |  _|   | | |  _| | |_) \___ \ 			//
// |  _ <| |___ / ___ \| |_| | |  __/ ___ \|  _ < / ___ \| |  | | |___  | | | |___|  _ < ___) |			//
// |_| \_|_____/_/   \_|____/  |_| /_/   \_|_| \_/_/   \_|_|  |_|_____| |_| |_____|_| \_|____/ 			//
//                                                                                           			//
//////////////////////////////////////////////////////////////////////////////////////////////////////////
(*
Check NC parameters available from MCReadParameter FB (17 in total)
See eRWParameter DUT for complete list or PLC OPEN documentation
To call all 17 from a single functionblock instance only 1 can be checked per cycle so there will be at minimum a 34 cycle delay checking each parameter
The MCReadParameter does also cover the functionality of MCReadBoolParameter so these booleans are separately converted from the MCReadParameter call
*)
MCReadParameter(Axis:=AxisController.AXIS,ParameterNumber:=iParam);
IF MCReadParameter.Valid THEN
	MCReadParameter.Enable:=FALSE;
	AxisController.fParameters[iParam]:=MCReadParameter.Value;
	iParam:= iParam+1;
	IF iParam>17 THEN
		iParam:=1;
	END_IF
ELSE
	MCReadParameter.Enable:=TRUE;
END_IF

//Convert LREALS to BOOLS


IF AxisController.fParameters[eRWParameter.EnableLimitPos]=1 THEN
	AxisController.bSoftLimPosEn:=TRUE;
ELSE
	AxisController.bSoftLimPosEn:=FALSE;
END_IF
IF AxisController.fParameters[eRWParameter.EnableLimitNeg]=1 THEN
	AxisController.bSoftLimNegEn:=TRUE;
ELSE
	AxisController.bSoftLimNegEn:=FALSE;
END_IF
IF AxisController.fParameters[eRWParameter.EnablePosLagMonitoring]=1 THEN
	AxisController.bPosLagEn:=TRUE;
ELSE
	AxisController.bPosLagEn:=FALSE;
END_IF

//////////////////////////////////////////////////////////////////////////////////////////////////////////
//  __  __  ____   _____ _   _ _   _  ____ _____ ___ ___  _   _    ____    _    _     _     ____  		//
// |  \/  |/ ___| |  ___| | | | \ | |/ ___|_   _|_ _/ _ \| \ | |  / ___|  / \  | |   | |   / ___| 		//
// | |\/| | |     | |_  | | | |  \| | |     | |  | | | | |  \| | | |     / _ \ | |   | |   \___ \ 		//
// | |  | | |___  |  _| | |_| | |\  | |___  | |  | | |_| | |\  | | |___ / ___ \| |___| |___ ___) |		//
// |_|  |_|\____| |_|    \___/|_| \_|\____| |_| |___\___/|_| \_|  \____/_/   \_|_____|_____|____/ 		//
//                                         																//                                                      
//////////////////////////////////////////////////////////////////////////////////////////////////////////
(*
Call MC Function Blocks and clear execute signals
Any MC function blocks added to the state machine must be called here with the given format.
Some FBs have slightly differing structures so these should aim to conform to the existing structure
Function blocks will hold done and error signals for 1 cycle with no execute held
*)
MCReadParameter(Axis:=AxisController.Axis);	//Reading in motion parameters, using one functionblock for all params means need to disable

MCReset(Axis:=AxisController.Axis);
MCReset.Execute:=FALSE;

MCWriteParameter(Axis:=AxisController.Axis);
MCWriteParameter.Execute:=FALSE;

MCWriteBoolParameter(Axis:=AxisController.Axis);
MCWriteBoolParameter.Execute:=FALSE;

MCSetPosition(Axis:=AxisController.Axis);
MCSetPosition.Execute:=FALSE;

MCMoveAbsolute(Axis:=AxisController.Axis);
MCMoveAbsolute.Execute:=FALSE;

MCMoveRelative(Axis:=AxisController.Axis);
MCMoveRelative.Execute:=FALSE;

MCGearIn(Slave:=AxisController.Axis, Master:=GVL.axes[AxisController.masterAxis].Axis);
MCGearIn.Execute:=FALSE;

MCGearInMultiMaster(Master1:=GVL.axes[AxisController.masterAxes[1].i].Axis,Master2:=GVL.axes[AxisController.masterAxes[2].i].Axis,Master3:=GVL.axes[AxisController.masterAxes[3].i].Axis,Master4:=GVL.axes[AxisController.masterAxes[4].i].Axis,Slave:=AxisController.Axis);
MCGearInMultiMaster.Enable:=FALSE;	//NOT EXECUTE AS FB ALLOWS CONTINUAL UPDATING OF RATIOS WHILST ENABLED

MCGearOut(Slave:=AxisController.Axis);
MCGearOut.Execute:=FALSE;

MCJog(Axis:=AxisController.Axis);
MCJog.JogBackwards:=FALSE;
MCJog.JogForward:=FALSE;

MCStepAbsoluteSwitch(Axis:=AxisController.Axis,Parameter:=MCHomingParameter);
MCStepAbsoluteSwitch.Execute:=FALSE;


MCFinishHoming(Axis:=AxisController.Axis,Parameter:=MCHomingParameter);
MCFinishHoming.Execute:=FALSE;

MCMoveVelocity(Axis:=AxisController.Axis);
MCMoveVelocity.Execute:=FALSE;

MCStop(Axis:=AxisController.Axis);
MCStop.Execute:=FALSE;

//////////////////////////////////////////////////////////////////////////////////////////////////////////////////////////////////////////////
//   ____ ___  __  __ __  __    _    _   _ ____     ____    _    ____  _____   ____ _____  _  _____ _____ __  __ _____ _   _ _____ ____ 	// 
//  / ___/ _ \|  \/  |  \/  |  / \  | \ | |  _ \   / ___|  / \  / ___|| ____| / ___|_   _|/ \|_   _| ____|  \/  | ____| \ | |_   _/ ___| 	//
// | |  | | | | |\/| | |\/| | / _ \ |  \| | | | | | |     / _ \ \___ \|  _|   \___ \ | | / _ \ | | |  _| | |\/| |  _| |  \| | | | \___ \ 	//
// | |__| |_| | |  | | |  | |/ ___ \| |\  | |_| | | |___ / ___ \ ___) | |___   ___) || |/ ___ \| | | |___| |  | | |___| |\  | | |  ___) |	//
//  \____\___/|_|  |_|_|  |_/_/   \_|_| \_|____/   \____/_/   \_|____/|_____| |____/ |_/_/   \_|_| |_____|_|  |_|_____|_| \_| |_| |____/	//
//																																			//
//////////////////////////////////////////////////////////////////////////////////////////////////////////////////////////////////////////////

(*
Internal statemachine to handle motion control flow and logic.
Functions are NOT called in this statemachine, these just update values given to the state machine. This was the method recommended by Beckhoff
The following basic wrapper should be used for adding new function blocks. Any that do not conform to this should be modified to conform
Notably some FBs have no .Done but do have .Active
	
	mcFunctionBlock.Execute		:=AxisController.bExecute;
	mcFunctionBlock.misc1..n	:=AxisController.misc1..n;
	
	bDone:=mcFunctionBlock.Done;
	AxisController.bBusy:= mcFunctionBlock.Busy;
	
	If mcFunctionBlock.Error THEN
		AxisController.bError:=TRUE;
		AxisController.iErrorID:= mcFunctionBlock.ErrorID;
	END_IF
	IF NOT mcFunctionBlock.Busy THEN
		eCommandLatched:=eMcCommand.Idle;
	END_IF
	
Function block specific parameters should be added to the ST_AxisControl if not already listed
eCommandLatched is currently being used to hold control flow logic so that users cannot send new commands until previous ones have complete.
This will definitely need to be modified to allow buffering in the future and to allow stop/halt commands 
but I haven't looked in to the best way to do this yet.	

It may be that it doesn't matter if it is latched at all as we can rely on waiting for the done signal before sending subsequent commands if it really matters
*)
//If we're not doing anything or have just done something we no longer latch on the given command
eCommandLatched:=AxisController.eCommand;

CASE eCommandLatched OF
	
	eMcCommand.Idle:
		AxisController.bBusy	:=FALSE;
		AxisController.bExecute	:=FALSE;
///////////////////////////////////////////////////////////////////////////////////////////////////////////////////////////////	
	eMcCommand.Reset:
		AxisController.bError	:=FALSE;
		MCReset.Execute:=AxisController.bReset;
		
		bDone:=McReset.Done;
		AxisController.bBusy:=MCReset.Busy;
		IF MCReset.Error THEN
			AxisController.bError:=TRUE;
			AxisController.iErrorID:=MCReset.ErrorID;	
		END_IF
		IF NOT MCReset.Busy THEN
			eCommandLatched:=eMcCommand.Idle;
			AxisController.bReset:=FALSE;
		END_IF
///////////////////////////////////////////////////////////////////////////////////////////////////////////////////////////////
	eMcCommand.WriteParameter:		
		MCWriteParameter.Execute:=AxisController.bExecute;
		MCWriteParameter.ParameterNumber:=AxisController.iParameterIndex;
		MCWriteParameter.Value:=AxisController.fParameterValue;
		
		bDone:=MCWriteParameter.Done;
		AxisController.bBusy:= MCWriteParameter.Busy;
		
		IF MCWriteParameter.Error THEN
			AxisController.bError:=TRUE;
			AxisController.iErrorID:=MCWriteParameter.ErrorID;	
		END_IF	
		IF NOT MCWriteParameter.Busy THEN
			eCommandLatched:=eMcCommand.Idle;
		END_IF			
///////////////////////////////////////////////////////////////////////////////////////////////////////////////////////////////
	eMcCommand.WriteBoolParameter:	
		MCWriteBoolParameter.Execute:=AxisController.bExecute;
		MCWriteBoolParameter.ParameterNumber:=AxisController.iParameterIndex;
		MCWriteBoolParameter.Value:=AxisController.bInput;
		
		bDone:=MCWriteBoolParameter.Done;
		AxisController.bBusy:=MCWriteBoolParameter.Busy;
		
		IF MCWriteBoolParameter.Error THEN
			AxisController.bError:= TRUE;
			AxisController.iErrorID:=MCWriteBoolParameter.ErrorID;
		END_IF			
		IF NOT MCWriteBoolParameter.Busy THEN
			eCommandLatched:=eMcCommand.Idle;
		END_IF	
///////////////////////////////////////////////////////////////////////////////////////////////////////////////////////////////
	eMcCommand.SetPosition:	
		MCSetPosition.Execute:=AxisController.bExecute;
		MCSetPosition.Position:=AxisController.fPosition;
		
		AxisController.bBusy:=MCSetPosition.Busy;
		bDone:=MCSetPosition.Done;
		
		IF MCSetPosition.Error THEN
			AxisController.bError:=TRUE;
			AxisController.iErrorID:= MCSetPosition.ErrorID;
		END_IF
		IF NOT MCSetPosition.Busy THEN
			eCommandLatched:=eMcCommand.Idle;
		END_IF
///////////////////////////////////////////////////////////////////////////////////////////////////////////////////////////////
	eMcCommand.MoveAbsolute:	
		MCMoveAbsolute.Execute:=AxisController.bExecute;
		MCMoveAbsolute.Position:=AxisController.fPosition;
		MCMoveAbsolute.Velocity:=AxisController.fVelocity;
		MCMoveAbsolute.Acceleration:=AxisController.fAcceleration;
		MCMoveAbsolute.Deceleration:=AxisController.fDeceleration;
		MCMoveAbsolute.Jerk:=0;
		//MCMoveAbsolute.BufferMode:=MC_BufferMode.MC_Buffered;
		
		bDone:=MCMoveAbsolute.Done;
		AxisController.bBusy:=MCMoveAbsolute.Busy;
		
		IF MCMoveAbsolute.Error THEN
			AxisController.bError:=TRUE;
			AxisController.iErrorID:=MCMoveAbsolute.ErrorID;
		END_IF
		IF NOT MCMoveAbsolute.Busy THEN
			eCommandLatched:=eMcCommand.Idle;
		END_IF
///////////////////////////////////////////////////////////////////////////////////////////////////////////////////////////////
	eMcCommand.MoveRelative:		
		MCMoveRelative.Execute:=AxisController.bExecute;
		MCMoveRelative.Distance:=AxisController.fDistance;
		MCMoveRelative.Velocity:=AxisController.fVelocity;
		MCMoveRelative.Acceleration:=AxisController.fAcceleration;
		MCMoveRelative.Deceleration:=AxisController.fDeceleration;
		MCMoveRelative.Jerk:=0;
		//MCMoveRelative.BufferMode:=MC_BufferMode.MC_Buffered;
		
		bDone:=MCMoveRelative.Done;
		AxisController.bBusy:=MCMoveRelative.Busy;
		
		IF MCMoveRelative.Error THEN
			AxisController.bError:=TRUE;
			AxisController.iErrorID:=MCMoveRelative.ErrorID;
		END_IF
		IF NOT MCMoveRelative.Busy THEN
			eCommandLatched:=eMcCommand.Idle;
		END_IF		
///////////////////////////////////////////////////////////////////////////////////////////////////////////////////////////////
	eMcCommand.GearIn:
		//Dependent on +ve or -ve gear ratio determines whether to link Fw to Fw and Bw to Bw or Fw to Bw and Bw to Fw
		IF AxisController.fGearRatioNum>0 THEN
			Limits.coupledFwLimit[GVL.iAxis][1].eLimitType:=eLimitCoupling.FwSw;		
			Limits.coupledBwLimit[GVL.iAxis][1].eLimitType:=eLimitCoupling.BwSw;				
		END_IF
		IF AxisController.fGearRatioNum<0 THEN
			Limits.coupledFwLimit[GVL.iAxis][1].eLimitType:=eLimitCoupling.BwSw;
			Limits.coupledBwLimit[GVL.iAxis][1].eLimitType:=eLimitCoupling.FwSw;		
		END_IF
		Limits.coupledFwLimit[GVL.iAxis][1].iMasterAxis:=AxisController.masterAxis;
		Limits.coupledBwLimit[GVL.iAxis][1].iMasterAxis:=AxisController.masterAxis;
		
		MCGearIn.Execute:=AxisController.bExecute;
		MCGearIn.RatioNumerator:=AxisController.fGearRatioNum;
		MCGearIn.RatioDenominator:=AxisController.iGearRatioDen;
		
		bDone:=McGearIn.InGear;
		AxisController.bBusy:=MCGearIn.Busy;
		
		IF MCGearIn.Error THEN
			AxisController.bError:=TRUE;
			AxisController.iErrorID:=MCGearIn.ErrorID;
		END_IF		
		IF NOT MCGearIn.Busy THEN
			eCommandLatched:=eMcCommand.Idle;
		END_IF
///////////////////////////////////////////////////////////////////////////////////////////////////////////////////////////////
	eMcCommand.GearInMultiMaster:		
		//Set up limits
		FOR iMasterIndex:=1 TO GVL.axisCoupleMax DO
			IF AxisController.masterAxes[iMasterIndex].ratio>0 THEN
				Limits.coupledFwLimit[GVL.iAxis][iMasterIndex+1].eLimitType:=eLimitCoupling.FwSw;				
				Limits.coupledBwLimit[GVL.iAxis][iMasterIndex+1].eLimitType:=eLimitCoupling.BwSw;				
			END_IF
			IF AxisController.masterAxes[iMasterIndex].ratio<0 THEN
				Limits.coupledFwLimit[GVL.iAxis][iMasterIndex+1].eLimitType:=eLimitCoupling.BwSw;
				Limits.coupledBwLimit[GVL.iAxis][iMasterIndex+1].eLimitType:=eLimitCoupling.FwSw;
			END_IF
			Limits.coupledFwLimit[GVL.iAxis][iMasterIndex+1].iMasterAxis:=AxisController.masterAxes[iMasterIndex].i;
			Limits.coupledBwLimit[GVL.iAxis][iMasterIndex+1].iMasterAxis:=AxisController.masterAxes[iMasterIndex].i;
		END_FOR
		

		
		(*	Issue with this MC block (other than everything...) is that it doesn't conform to the standard and use an execute signal. The execute
			signal in any other block determines that when it is high one of either error,done,busy must be on. That is not the case with this block
			what happens is it triggers, doesn't register a busy and so immediately clears as done. If has been modified to conform.
		*)
		MCGearInMultiMaster.Enable:=AxisController.bExecute;
		MCGearInMultiMaster.GearRatio1:=AxisController.masterAxes[1].ratio;
		MCGearInMultiMaster.GearRatio2:=AxisController.masterAxes[2].ratio;
		MCGearInMultiMaster.GearRatio3:=AxisController.masterAxes[3].ratio;
		MCGearInMultiMaster.GearRatio4:=AxisController.masterAxes[4].ratio;
		
		AxisController.bBusy:=MCGearInMultiMaster.Busy;
		IF MCGearInMultiMaster.Enable THEN
			AxisController.bBusy:=TRUE;	//busy does not go immediately high when enable high 
			bDone:=FALSE;
		END_IF

		bDone:=MCGearInMultiMaster.InGear;	
		IF MCGearInMultiMaster.Error THEN
			AxisController.bError:=TRUE;
			AxisController.iErrorID:=MCGearInMultiMaster.ErrorID;
		END_IF
		IF NOT MCGearInMultiMaster.Busy THEN
			eCommandLatched:=eMcCommand.Idle;
		END_IF
///////////////////////////////////////////////////////////////////////////////////////////////////////////////////////////////
	eMcCommand.GearOut:		
		//Gearout - remove all masters from slave
		FOR iMasterIndex:=1 TO 5 DO
				Limits.coupledFwLimit[GVL.iAxis][iMasterIndex].eLimitType:=eLimitCoupling.None;
				Limits.coupledBwLimit[GVL.iAxis][iMasterIndex].eLimitType:=eLimitCoupling.None;
		END_FOR		
	
		MCGearOut.Execute:=AxisController.bExecute;
		
		AxisController.bBusy:=MCGearOut.Busy;
		bDone:=MCGearOut.Done;
		IF MCGearOut.Error THEN
			AxisController.bError:=TRUE;
			AxisController.iErrorID:=MCGearOut.ErrorID;
		END_IF
		IF NOT MCGearOut.Busy THEN
			eCommandLatched:=eMcCommand.Idle;
		END_IF
	///////////////////////////////////////////////////////////////////////////////////////////////////////////////////////////////			
	eMcCommand.Jog:
		MCJog.JogForward:=AxisController.bJogForward;
		MCJog.JogBackwards:=AxisController.bJogBackward;
		
		bDone:=MCJog.Done;
		
		IF MCJog.Error THEN
			AxisController.bError:=TRUE;
			AxisController.iErrorID:=MCJog.ErrorID;
		END_IF
		IF NOT MCJog.Busy THEN
			eCommandLatched:=eMcCommand.Idle;
		END_IF
	///////////////////////////////////////////////////////////////////////////////////////////////////////////////////////////////	
	eMcCommand.HomeStepAbsoluteSwitch:
		//Issue: If execute not held high the function will not reverse on its own to find the abs switch when hitting a limit
		//You have to reissue the command. I want to try and keep bExecute high
		IF (NOT Limits.FwLimit[GVL.iAxis]) OR (NOT Limits.BwLimit[GVL.iAxis]) THEN
			MCStepAbsoluteSwitch.Execute:=TRUE;
		ELSE	
			MCStepAbsoluteSwitch.Execute:=AxisController.bExecute;
		END_IF
	
		MCStepAbsoluteSwitch.Direction:= AxisController.mcHomeDirection;
		MCStepAbsoluteSwitch.SwitchMode:=AxisController.mcSwitchMode;
		MCStepAbsoluteSwitch.ReferenceSignal:=AxisController.mcSignalRef;
		MCStepAbsoluteSwitch.Velocity:=AxisController.fHomeVelocity;
		MCStepAbsoluteSwitch.Acceleration:=0;
		MCStepAbsoluteSwitch.Deceleration:=0;
		MCStepAbsoluteSwitch.Jerk:=0;
		MCStepAbsoluteSwitch.TorqueLimit:=AxisController.fHomeTorque;
		MCStepAbsoluteSwitch.SetPosition:=AxisController.fHomePosition;
		MCStepAbsoluteSwitch.TimeLimit:=AxisController.tHomeTimeLimit;
		MCStepAbsoluteSwitch.DistanceLimit:=AxisController.fHomeDistanceLimit;
		MCStepAbsoluteSwitch.PositiveLimitSwitch:= NOT Limits.FwLimit[GVL.iAxis];	//Step FB has R_TRIG behaviour but limits set as Normally Closed so logic is inverted
		MCStepAbsoluteSwitch.NegativeLimitSwitch:= NOT Limits.BwLimit[GVL.iAxis];	//Step FB has R_TRIG behaviour but limits set as Normally Closed so logic is inverted
		MCStepAbsoluteSwitch.BufferMode:=AxisController.buffer;
		StOptions4.DisableDriveAccess:=TRUE;		//Testing required with hardware. This step may be redundant.
		MCStepAbsoluteSwitch.Options:=StOptions4;
		
		bDone:=MCStepAbsoluteSwitch.Done;
		AxisController.bBusy:=MCStepAbsoluteSwitch.Busy;
		
		IF MCStepAbsoluteSwitch.Error THEN
			AxisController.bError:=TRUE;
			AxisController.iErrorID:=MCStepAbsoluteSwitch.ErrorID;
		END_IF
		IF NOT MCStepAbsoluteSwitch.Busy THEN
			eCommandLatched:=eMcCommand.Idle;
		END_IF
	///////////////////////////////////////////////////////////////////////////////////////////////////////////////////////////////	
	eMcCommand.HomeFinish:
		MCFinishHoming.Execute:=AxisController.bExecute;
		MCFinishHoming.Distance:=AxisController.fHomeDistance;
		MCFinishHoming.Velocity:=AxisController.fHomeVelocity;
		
		StOptions2.DisableDriveAccess:=TRUE;	//Testing required with hardware. This step may be redundant.
		MCFinishHoming.Options:=StOptions2;
		
		bDone:=MCFinishHoming.Done;
		AxisController.bBusy:=MCFinishHoming.Busy;
		
		IF MCFinishHoming.Error THEN
			AxisController.bError:=TRUE;
			AxisController.iErrorID:=MCFinishHoming.ErrorID;
		END_IF
		IF NOT MCFinishHoming.Busy THEN
			eCommandLAtched:=eMcCommand.Idle;
		END_IF
	///////////////////////////////////////////////////////////////////////////////////////////////////////////////////////////////	
	eMcCommand.MoveVelocity:
		MCMoveVelocity.Execute:=AxisController.bExecute;
		MCMoveVelocity.Acceleration:=AxisController.fAcceleration;
		MCMoveVelocity.Deceleration:=AxisController.fDeceleration;
		
		//Simple logic to allow negative velocity inputs rather than having to set the direction object
		IF AxisController.fVelocity>= 0 THEN
			MCMoveVelocity.Velocity:=AxisController.fVelocity;
			MCMoveVelocity.Direction:= MC_Positive_Direction;
		ELSE
			MCMoveVelocity.Velocity:=ABS(AxisController.fVelocity);
			MCMoveVelocity.Direction:= MC_Negative_Direction;
		END_IF
		
		bDone:=MCMoveVelocity.InVelocity;
		AxisController.bBusy:=MCMoveVelocity.Busy;
		
		IF MCMoveVelocity.Error THEN
			AxisController.bError:=TRUE;
			AxisController.iErrorID:=MCMoveVelocity.ErrorID;
		END_IF
		IF NOT MCMoveVelocity.Busy THEN
			eCommandLatched:=eMcCommand.Idle;
		END_IF
	///////////////////////////////////////////////////////////////////////////////////////////////////////////////////////////////	
	eMcCommand.Stop:
		McStop.Execute:=AxisController.bExecute;
		McStop.Deceleration:=AxisController.fDeceleration;
		McStop.Jerk:=0;
		
		bDone:=McStop.Done;
		AxisController.bBusy:=McStop.Busy;
		
		IF MCStop.Error THEN
			AxisController.bError:= TRUE;
			AxisController.iErrorID:=MCStop.ErrorId;
		END_IF
		IF	NOT MCStop.Busy THEN
			eCommandLatched:=eMcCommand.Idle;
		END_IF

		
END_CASE

////////////////////////////////////////// 
//  _____ _        _    ____ ____  		//
// |  ___| |      / \  / ___/ ___| 		//
// | |_  | |     / _ \| |  _\___ \ 		//
// |  _| | |___ / ___ | |_| |___) |		//
// |_|   |_____/_/   \_\____|____/ 		//
//                                		//
//////////////////////////////////////////
AxisController.bMoving:=AxisController.Axis.Status.Moving;	
AxisController.bExecute:=FALSE;

(*
As we never hold Execute high, the done signal from each function block will only stay on for 1 cycle tick
The following logic just uses an SR latch to hold this done signal TRUE until it is cleared either by an error or the axis going busy

Errors are always latched as they are only ever set by a FB error and cleared by a reset command
*)
doneLatch(SET1:=bDone,RESET:=(AxisController.bBusy OR AxisController.bError));
AxisController.bDone:=doneLatch.Q1;

END_FUNCTION_BLOCK

// ---- GlobalTextList.TcGTLO
TEXTLIST GlobalTextList
  619 = ' ADVANCED HOMING '
  800 = ' DISCRETE MOVES '
  922 = ' GEARING '
  86 = ' MULTI-GEARING '
  176 = ' Parameters '
  807 = ' POWER '
  779 = ' Simulation '
  243 = '%2.2f'
  808 = '%3.2f'
  803 = '%4.2f'
  926 = '%d'
  445 = '%s'
  244 = '+'
  245 = '-'
  801 = 'ABS.MOVE'
  783 = 'Absolute Flag High Position'
  784 = 'Absolute Flag Low Position'
  822 = 'ActualVelocity'
  449 = 'Adv. Homing'
  441 = 'AXIS BUSY'
  806 = 'AXIS NAME:'
  804 = 'AXIS SELECTION:'
  810 = 'BW'
  452 = 'BW ENABLED'
  444 = 'CALIBRATED'
  178 = 'Cmd Position:'
  823 = 'CommandedVelocity'
  927 = 'DEN.'
  102 = 'Disable MC'
  787 = 'Distance:'
  443 = 'DONE'
  809 = 'EN'
  101 = 'ENABLE H'
  100 = 'ENABLE V'
  442 = 'ERROR'
  788 = 'FINISH HOMING'
  811 = 'FW'
  453 = 'FW ENABLED'
  928 = 'GEAR IN'
  929 = 'GEAR OUT'
  923 = 'GEARED'
  447 = 'Gearing'
  407 = 'HC:'
  406 = 'HG:'
  781 = 'High Limit Position'
  604 = 'I/O'
  782 = 'Low Limit Position'
  87 = 'MASTER1:'
  89 = 'MASTER2:'
  90 = 'MASTER3:'
  727 = 'MASTER4:'
  924 = 'MASTER:'
  824 = 'MaxAccelerationAppl'
  981 = 'MaxAccelerationSystem'
  622 = 'MaxDecelerationAppl'
  825 = 'MaxDecelerationSystem'
  623 = 'MaxJerkAppl'
  826 = 'MaxJerkSystem'
  819 = 'MaxPositionLag'
  821 = 'MaxVelocityAppl'
  820 = 'MaxVelocitySystem'
  925 = 'NUM.'
  448 = 'Parameters'
  88 = 'RATIO:'
  451 = 'Read Position:'
  802 = 'REL.MOVE'
  446 = 'RESET'
  817 = 'SET'
  786 = 'Set Position:'
  789 = 'Simulate AbsSw/Pulse'
  780 = 'Simulated Axis'
  450 = 'Simulation'
  602 = 'Single Axis'
  603 = 'Slit Set'
  620 = 'STEP ABS SW'
  455 = 'STOP'
  827 = 'SWLimitNeg:'
  177 = 'SWLimitPos:'
  818 = 'Toggle'
  247 = 'VC:'
  805 = 'Velocity'
  454 = 'VELOCITY MOVE'
  785 = 'Velocity:'
  246 = 'VG:'
END_TEXTLIST

// ---- VISUs/Main.TcVIS
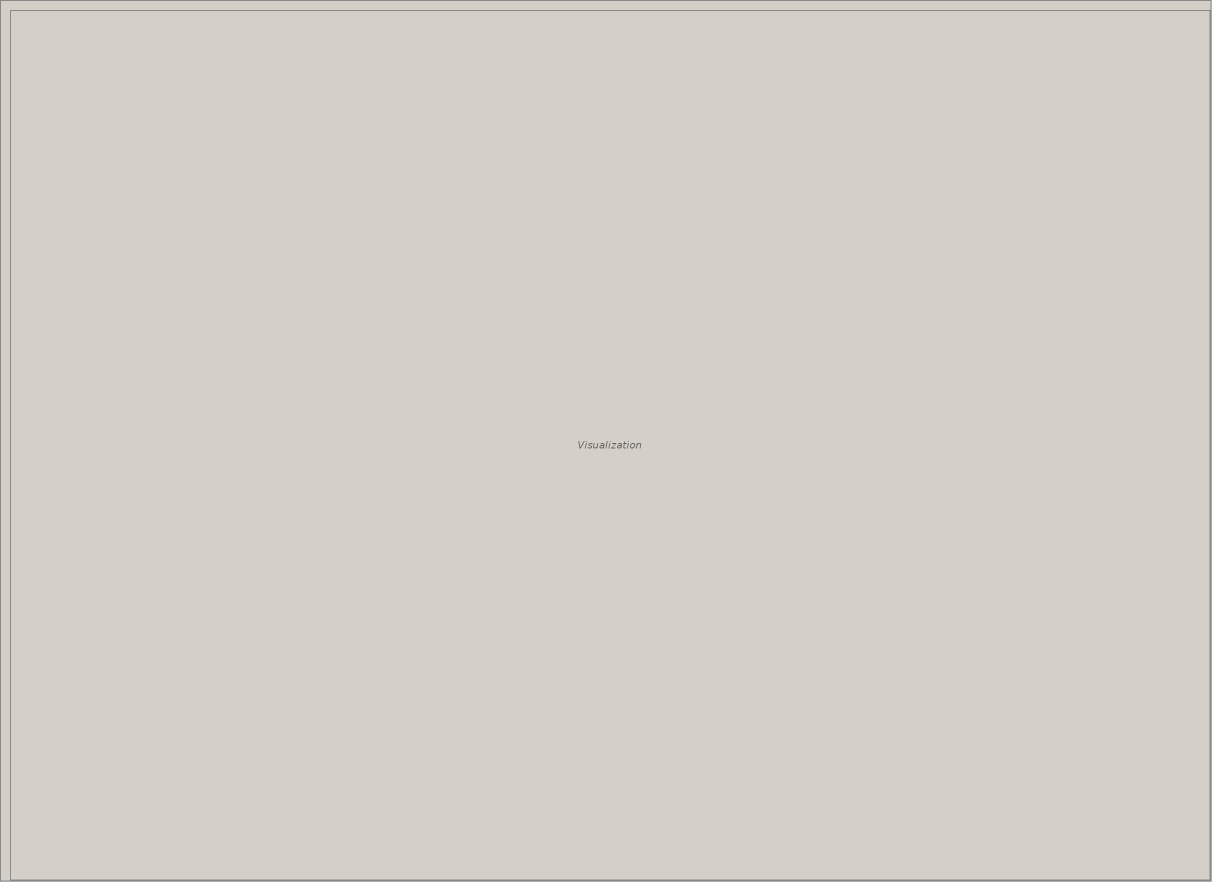
VISUALIZATION Main  // 1212x882
    TabControl (10,10 1200x870)
        shows Visualization()
        shows SlitSet()
        shows IO()
        [0]: TabTitle=Single Axis
        [1]: TabTitle=Slit Set
END_VISUALIZATION

// ---- VISUs/Panels/Visualization.TcVIS
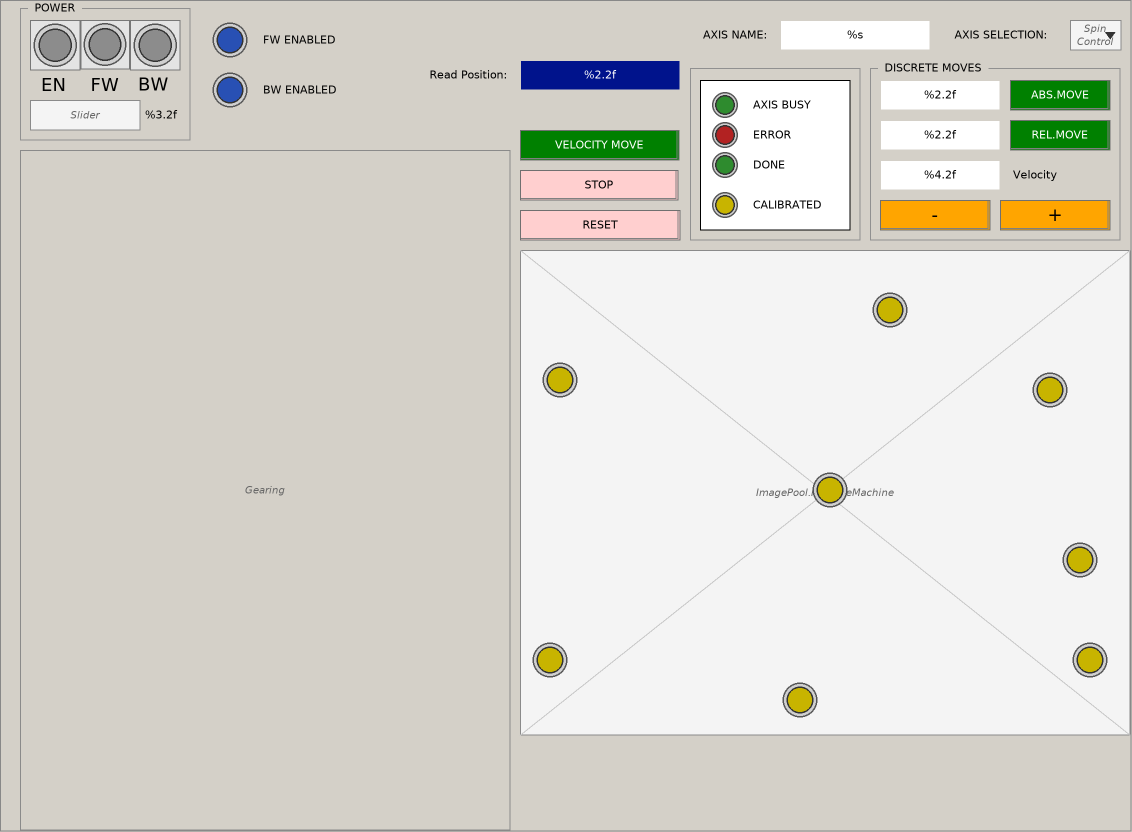
VISUALIZATION Visualization  // 1132x832
    GroupBox (870,60 250x180), "DISCRETE MOVES"
        Textfield (10,20 120x30), "%2.2f", text variable: GVL.axes[MAIN.hmiAxisSelect].fPosition
            OnMouseClick: write GVL.axes[MAIN.hmiAxisSelect].fPosition via Default
        Button (140,20 100x30), "ABS.MOVE"
            OnMouseClick: execute { GVL.axes[MAIN.hmiAxisSelect].eCommand:=eMcCommand.MoveAbsolute; GVL.axes[MAIN.hmiAxisSelect].bEXECUTE:= TRUE; }
        Textfield (10,60 120x30), "%2.2f", text variable: GVL.axes[MAIN.hmiAxisSelect].fDistance
            OnMouseClick: write GVL.axes[MAIN.hmiAxisSelect].fDistance via Default
        Button (140,60 100x30), "REL.MOVE", input disabled if: GVL.axes[MAIN.hmiAxisSelect].iAxisState=500
            OnMouseClick: execute { GVL.axes[MAIN.hmiAxisSelect].eCommand:=eMcCommand.MoveRelative; GVL.axes[MAIN.hmiAxisSelect].bEXECUTE:= TRUE; }
        Button (10,140 110x30), "-"
            tap GVL.axes[MAIN.hmiAxisSelect].bJogBackward
            OnMouseClick: execute { GVL.axes[MAIN.hmiAxisSelect].eCommand:=eMcCommand.Jog; }
        Button (130,140 110x30), "+"
            tap GVL.axes[MAIN.hmiAxisSelect].bJogForward
            OnMouseClick: execute { GVL.axes[MAIN.hmiAxisSelect].eCommand:=eMcCommand.Jog; }
        Textfield (10,100 120x30), "%4.2f", text variable: GVL.axes[MAIN.hmiAxisSelect].fVelocity
            OnMouseClick: write GVL.axes[MAIN.hmiAxisSelect].fVelocity via Default
    Textfield (520,60 160x30), "%2.2f", text variable: GVL.axes[MAIN.hmiAxisSelect].Axis.NcToPlc.ActPos
    SpinControl (1070,20 51x30), variable: MAIN.hmiAxisSelect
        p651134158: GVL.axisNumMax
    Textfield (930,20 120x30), "AXIS SELECTION:", text variable: MAIN.hmiAxisSelect
    Textfield (1010,160 100x30), "Velocity", text variable: MAIN.hmiAxisSelect
    Textfield (650,20 120x30), "AXIS NAME:"
    GroupBox (20,0 170x140), "POWER"
        PushSwitchLed (110,20 50x50), variable: Limits.BwLimit[MAIN.hmiAxisSelect], behaviour: TOGGLE, style: Switch-PushSwitchLed-Gray
        Slider (10,100 110x30), variable: GVL.axes[MAIN.hmiAxisSelect].fOverride, scale 0..100
        Textfield (120,100 40x30), "%3.2f", text variable: GVL.axes[MAIN.hmiAxisSelect].fOverride
        Label (10,70 47x30), "EN"
        Label (110,70 47x29), "BW"
        PushSwitchLed (60,20 50x49), variable: Limits.FwLimit[MAIN.hmiAxisSelect], behaviour: TOGGLE, style: Switch-PushSwitchLed-Gray
        Label (60,70 50x30), "FW"
        PushSwitchLed (10,20 50x50), variable: GVL.axes[MAIN.hmiAxisSelect].bEnable, behaviour: TOGGLE, style: Switch-PushSwitchLed-Gray
    GroupBox (690,60 170x180)
        Rectangle (10,20 150x150)
        Lamp1 (20,30 30x30), variable: GVL.axes[MAIN.hmiAxisSelect].bBusy, style: Lamp-Lamp1-Green
        Lamp1 (20,60 30x30), variable: GVL.axes[MAIN.hmiAxisSelect].bError, style: Lamp-Lamp1-Red
        Lamp1 (20,90 30x30), variable: GVL.axes[MAIN.hmiAxisSelect].bDone, style: Lamp-Lamp1-Green
        Textfield (60,30 90x30), "AXIS BUSY", text variable: MAIN.hmiAxisSelect
        Textfield (60,60 90x30), "ERROR", text variable: MAIN.hmiAxisSelect
        Textfield (60,90 90x30), "DONE", text variable: MAIN.hmiAxisSelect
        Lamp1 (20,130 30x30), variable: GVL.axes[MAIN.hmiAxisSelect].Axis.Status.Homed, style: Lamp-Lamp1-Yellow
        Textfield (60,130 90x30), "CALIBRATED", text variable: MAIN.hmiAxisSelect
    Textfield (780,20 150x30), "%s", text variable: GVL.axes[MAIN.hmiAxisSelect].sAxisName
        OnMouseClick: write GVL.axes[MAIN.hmiAxisSelect].sAxisName via Edit
    Button (520,210 160x30), "RESET"
        OnMouseClick: execute { GVL.axes[MAIN.hmiAxisSelect].eCommand:=eMcCommand.Reset; GVL.axes[MAIN.hmiAxisSelect].bReset:= TRUE; }
    Image (520,250 610x485), image: ImagePool.NCStateMachine
    Lamp1 (1070,640 40x40), variable: GVL.axes[MAIN.hmiAxisSelect].iAxisState=100, style: Lamp-Lamp1-Yellow
    Lamp1 (780,680 40x40), variable: GVL.axes[MAIN.hmiAxisSelect].iAxisState=200, style: Lamp-Lamp1-Yellow
    Lamp1 (530,640 40x40), variable: GVL.axes[MAIN.hmiAxisSelect].iAxisState=300, style: Lamp-Lamp1-Yellow
    Lamp1 (1060,540 40x40), variable: GVL.axes[MAIN.hmiAxisSelect].iAxisState=999, style: Lamp-Lamp1-Yellow
    Lamp1 (810,470 40x40), variable: GVL.axes[MAIN.hmiAxisSelect].iAxisState=700, style: Lamp-Lamp1-Yellow
    Lamp1 (1030,370 40x40), variable: GVL.axes[MAIN.hmiAxisSelect].iAxisState=600, style: Lamp-Lamp1-Yellow
    Lamp1 (540,360 40x40), variable: GVL.axes[MAIN.hmiAxisSelect].iAxisState=400, style: Lamp-Lamp1-Yellow
    Lamp1 (870,290 40x40), variable: GVL.axes[MAIN.hmiAxisSelect].iAxisState=500, style: Lamp-Lamp1-Yellow
    TabControl (20,150 490x680)
        shows Gearing()
        shows Parameters()
        shows Homing()
        shows AxisSimulation()
        [0]: TabTitle=Gearing
        [1]: TabTitle=Parameters
        [2]: TabTitle=Adv. Homing
        [3]: TabTitle=Simulation
    Textfield (390,60 120x30), "Read Position:"
    Lamp1 (210,20 40x40), variable: GVL.axes[MAIN.hmiAxisSelect].bFwEnabled, style: Lamp-Lamp1-Blue
    Lamp1 (210,70 40x40), variable: GVL.axes[MAIN.hmiAxisSelect].bBwEnabled, style: Lamp-Lamp1-Blue
    Textfield (260,70 120x40), "BW ENABLED", text variable: MAIN.hmiAxisSelect
    Textfield (260,20 120x40), "FW ENABLED", text variable: MAIN.hmiAxisSelect
    Button (520,130 159x30), "VELOCITY MOVE", input disabled if: GVL.axes[MAIN.hmiAxisSelect].iAxisState=500
        OnMouseClick: execute { GVL.axes[MAIN.hmiAxisSelect].eCommand:=eMcCommand.MoveVelocity; GVL.axes[MAIN.hmiAxisSelect].bEXECUTE:= TRUE; }
    Button (520,170 158x30), "STOP"
        OnMouseClick: execute { GVL.axes[MAIN.hmiAxisSelect].eCommand:=eMcCommand.Stop; GVL.axes[MAIN.hmiAxisSelect].bExecute:= TRUE; }
END_VISUALIZATION
